// TIA Portal V15.1 export
// export: Created 2024-06-21T08:40:52.6901426Z, ExportSetting WithDefaults, DisplayName Totally Integrated Automation Portal, DisplayVersion V15.1 Update 5, DisplayName TIA Portal Openness, DisplayVersion V15.1 Update 5, DisplayName SINAMICS Startdrive Advanced, DisplayVersion V15.1, DisplayName G130, G150, S120, S150, SINAMICS MV, S210, DisplayVersion V15.1, DisplayName G110M, G120, G120C, G120D, G120P, DisplayVersion V15.1, DisplayName STEP 7 Professional, DisplayVersion V15.1 Update 5, DisplayName STEP 7 Safety, DisplayVersion V15.1, DisplayName WinCC Professional, DisplayVersion V15.1 Update 5, DisplayName SIMATIC Visualization Architect, DisplayVersion V15.1
FUNCTION_BLOCK "LChangeOfState"   // FB2103, FBD
TITLE = LChangeOfState
{ S7_Optimized_Access := 'TRUE' }
AUTHOR : VCC
FAMILY : Function
VERSION : 0.1
// =============================================================================
// This Module Handles Change Of State
// ============================================================================
// stored: AutoNumber false, IsIECCheckEnabled false, IsRetainMemResEnabled false, MemoryReserve 100, SetENOAutomatically False, UDAEnableTagReadback false
   VAR_INPUT
      I_In { ExternalAccessible := 'False'; ExternalVisible := 'False'; ExternalWritable := 'False'} : Bool;   // Input
   END_VAR
   VAR_OUTPUT
      O_OutPut { ExternalAccessible := 'False'; ExternalVisible := 'False'; ExternalWritable := 'False'} : Bool;   // Output
   END_VAR
   VAR
      PosEdge { ExternalAccessible := 'False'; ExternalVisible := 'False'; ExternalWritable := 'False'} : Bool;   // Edge
      PosEdgeResult { ExternalAccessible := 'False'; ExternalVisible := 'False'; ExternalWritable := 'False'} : Bool;   // Result
      NegEdge { ExternalAccessible := 'False'; ExternalVisible := 'False'; ExternalWritable := 'False'} : Bool;   // Edge
      NegEdgeResult { ExternalAccessible := 'False'; ExternalVisible := 'False'; ExternalWritable := 'False'} : Bool;   // Result
   END_VAR
   VAR_TEMP   // added for the SCL form of the ladder/FBD networks
      _w1 : Bool;
      _w2 : Bool;
   END_VAR
BEGIN

REGION Network 1: **** 4.4 - Machine Status - Calculation **** Create Edge
   // Create Edge
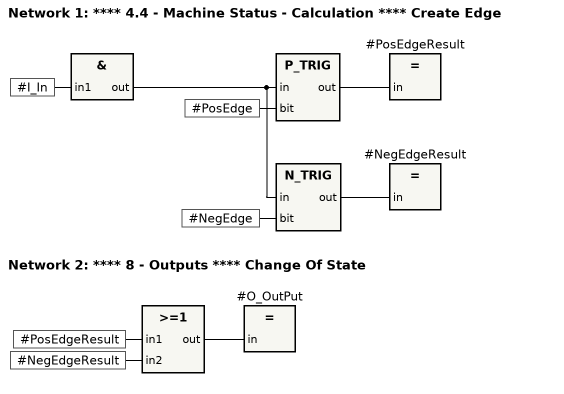
   #_w1 := #I_In AND NOT #PosEdge;   // rising edge
   #PosEdge := #I_In;
   #PosEdgeResult := #_w1;
   #_w2 := NOT #I_In AND #NegEdge;   // falling edge
   #NegEdge := #I_In;
   #NegEdgeResult := #_w2;
END_REGION

REGION Network 2: **** 8 - Outputs **** Change Of State
   // Change Of State
   #O_OutPut := #PosEdgeResult OR #NegEdgeResult;
END_REGION
END_FUNCTION_BLOCK
